Fanuc TP program (LS listing): LR_DPM_DEMO.LS

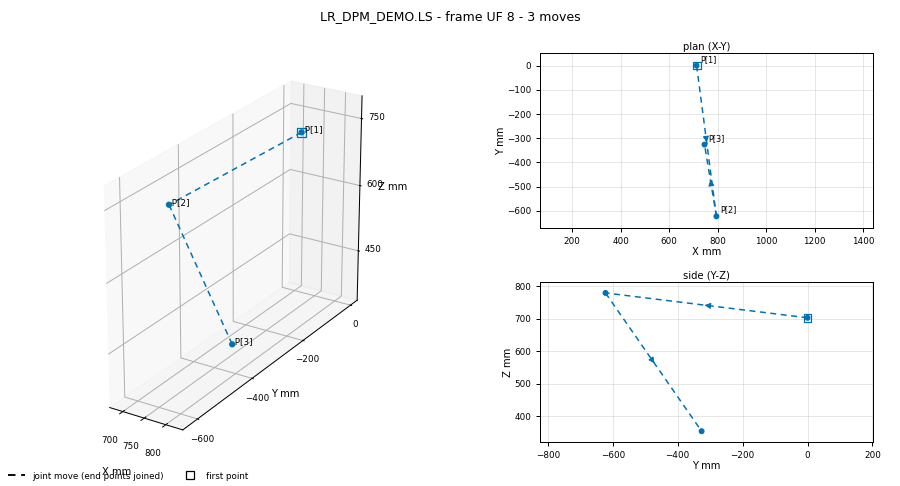
[picture p0: tool path of LR_DPM_DEMO.LS in frame UF 8, 3 of 6 moves have a stored position in this frame; points joined in program order, loops and branches not executed]
/PROG  LR_DPM_DEMO
/ATTR
OWNER		= MNEDITOR;
COMMENT		= "";
PROG_SIZE	= 1018;
CREATE		= DATE 24-09-14  TIME 15:04:56;
MODIFIED	= DATE 24-09-29  TIME 21:15:02;
FILE_NAME	= ;
VERSION		= 0;
LINE_COUNT	= 25;
MEMORY_SIZE	= 1298;
PROTECT		= READ_WRITE;
TCD:  STACK_SIZE	= 0,
      TASK_PRIORITY	= 50,
      TIME_SLICE	= 0,
      BUSY_LAMP_OFF	= 0,
      ABORT_REQUEST	= 0,
      PAUSE_REQUEST	= 0;
DEFAULT_GROUP	= 1,*,*,*,*;
CONTROL_CODE	= 00000000 00000000;
/MN
   1:  F[2]=(OFF) ;
   2:  F[3]=(OFF) ;
   3:  //F[4]=(OFF) ;
   4:  F[5]=(OFF) ;
   5:  RUN VS_CLIENT ;
   6:  WAIT (F[2]=ON)    ;
   7:J PR[6] 100% FINE    ;
   8:  !LOCAL REFERENCING ;
   9:J P[1] 100% FINE    ;
  10:  F[3]=(ON) ;
  11:  WAIT (F[3]=OFF)    ;
  12:J P[2] 100% FINE    ;
  13:  F[3]=(ON) ;
  14:  WAIT (F[3]=OFF)    ;
  15:J P[3] 100% FINE    ;
  16:  F[3]=(ON) ;
  17:  WAIT (F[3]=OFF)    ;
  18:  //WAIT (F[4]=ON)    ;
  19:  !DYN PATH MODIFICATION ;
  20:J PR[6] 100% FINE Offset,PR[7]    ;
  21:  F[5]=(ON) ;
  22:  Track DPM[1] ;
  23:L P[4] 10mm/sec FINE Offset,PR[7]    ;
  24:  Track End ;
  25:  F[5]=(OFF) ;
/POS
P[1]{
   GP1:
	UF : 8, UT : 1,		CONFIG : 'F U T, 0, 0, 0',
	X =   712.956  mm,	Y =      .000  mm,	Z =   703.315  mm,
	W =     -.000 deg,	P =   -88.036 deg,	R =  -180.000 deg
};
P[2]{
   GP1:
	UF : 8, UT : 1,		CONFIG : 'F U T, 0, 0, 0',
	X =   794.868  mm,	Y =  -622.273  mm,	Z =   779.892  mm,
	W =      .000 deg,	P =   -88.036 deg,	R =   180.000 deg
};
P[3]{
   GP1:
	UF : 8, UT : 1,		CONFIG : 'F U T, 0, 0, 0',
	X =   745.713  mm,	Y =  -326.209  mm,	Z =   354.014  mm,
	W =      .000 deg,	P =   -88.036 deg,	R =   179.999 deg
};
P[4]{
   GP1:
	UF : 8, UT : 1,		CONFIG : 'N U T, 0, 0, 0',
	X =   299.711  mm,	Y =     -.000  mm,	Z =   300.000  mm,
	W =   180.000 deg,	P =     -.000 deg,	R =     -.000 deg
};
/END
